// TIA Portal V19 export
TYPE "typePressureGuageRs485ControlNode"
TITLE = LBC_typeAnalogOutputControlNode
// Module related control node wrappe
// stored: Access Published
   STRUCT
      commands { ExternalVisible := 'False'} : "typePressureGuageRs485ControlNodeCommands";   // Module related commands from external systems
      monitoring { ExternalVisible := 'False'} : "typePressureGuageRs485ControlNodeMonitoring";   // Module related monitoring information
   END_STRUCT;
END_TYPE
